PROGRAM Mod101
VAR
	IO_f : ARRAY [1..16] OF IO_force;
	
	i: SINT;
END_VAR

	// 輸入模組1
	FOR i := 1 TO 16 DO
		IO_f[i](Raw_IO := EtherCAT.MainMod_1.Input[i], Out =>MainIO.IO101.In[i]);
	END_FOR
	
	
	MainIO.IO101_s.0 := IO_f[1].Out;
	MainIO.IO101_s.1 := IO_f[2].Out;
	MainIO.IO101_s.2 := IO_f[3].Out;
	MainIO.IO101_s.3 := IO_f[4].Out;
	MainIO.IO101_s.4 := IO_f[5].Out;
	MainIO.IO101_s.5 := IO_f[6].Out;
	MainIO.IO101_s.6 := IO_f[7].Out;
	MainIO.IO101_s.7 := IO_f[8].Out;
	MainIO.IO101_s.8 := IO_f[9].Out;
	MainIO.IO101_s.9 := IO_f[10].Out;
	MainIO.IO101_s.10 := IO_f[11].Out;
	MainIO.IO101_s.11 := IO_f[12].Out;
	MainIO.IO101_s.12 := IO_f[13].Out;
	MainIO.IO101_s.13 := IO_f[14].Out;
	MainIO.IO101_s.14 := IO_f[15].Out;
	MainIO.IO101_s.15 := IO_f[16].Out;
	
	MainIO.io101_f.0 := IO_f[1].ForceEnable;
	MainIO.io101_f.1 := IO_f[2].ForceEnable;
	MainIO.io101_f.2 := IO_f[3].ForceEnable;
	MainIO.io101_f.3 := IO_f[4].ForceEnable;
	MainIO.io101_f.4 := IO_f[5].ForceEnable;
	MainIO.io101_f.5 := IO_f[6].ForceEnable;
	MainIO.io101_f.6 := IO_f[7].ForceEnable;
	MainIO.io101_f.7 := IO_f[8].ForceEnable;
	MainIO.io101_f.8 := IO_f[9].ForceEnable;
	MainIO.io101_f.9 := IO_f[10].ForceEnable;
	MainIO.io101_f.10 := IO_f[11].ForceEnable;
	MainIO.io101_f.11 := IO_f[12].ForceEnable;
	MainIO.io101_f.12 := IO_f[13].ForceEnable;
	MainIO.io101_f.13 := IO_f[14].ForceEnable;
	MainIO.io101_f.14 := IO_f[15].ForceEnable;
	MainIO.io101_f.15 := IO_f[16].ForceEnable;

END_PROGRAM

(* stored: Version 1.1.0.1, ProductVersion 3.1.4024.15
   POU Mod101: Id {a2be50c4-ae63-4bed-9c22-38000c48133a}, SpecialFunc None *)
